// TwinCAT 3 PLC project PLC
// ProgramVersion: 3.1.4023.0
// libraries:
//   Tc2_Standard, * (Beckhoff Automation GmbH)
//   Tc2_System, * (Beckhoff Automation GmbH)
//   Tc3_Module, * (Beckhoff Automation GmbH)
// project tree:
//   / PlcTask.TcTTO
//   POUs/ MAIN.TcPOU
// real-time tasks:
//   TASK PlcTask: cycle T#4ms, priority 20, ADS port 350
// I/O:
//   DEVICE Device 1 (Profinet Controller), AmsNetId 5.24.131.22.2.1
//     tcpniodevice [Beckhoff Automation TwinCAT PLC PROFINET I/O Device with I/Os, V2.32, 1 port diagnostic supported TwinCAT PN Device]
//       modules: Term 1 (DAP Module), Term 2 (32 Byte In- and Output)
//   DEVICE Device 2 (TC3 EIP Scanner), AmsNetId 5.24.131.22.3.1
//     Box 2 (TC EtherNet/IP Slave) // <INFO> 172.16.17.2, Box 2 (TC EtherNet/IP Slave) (ProdCode: 6280, Rev: 3.01, Mac: 02:00:02:22:78:9c) </INFO> <EDS> C:\TwinCAT\3.1\Config\Io\EtherNetIP\TF6280.eds </EDS>
// variable links:
//   PLC Instance <-> Device 1 (Profinet Controller)/tcpniodevice
//     PlcTask Inputs/MAIN.arPNIn[{0..31}] <-> API/Term 2 (32 Byte In- and Output)/Subterm 4 (32 Byte In- and Output)/Inputs/1 Byte Input[{0..31}]  (32 links)
//     PlcTask Outputs/MAIN.arPNOut[{0..31}] <-> API/Term 2 (32 Byte In- and Output)/Subterm 4 (32 Byte In- and Output)/Outputs/1 Byte Output[{0..31}]  (32 links)
//   PLC Instance <-> Device 2 (TC3 EIP Scanner)/Box 2 (TC EtherNet/IP Slave)
//     PlcTask Inputs/MAIN.arEIPIn[{0..31}] <-> Connection 1 (Input/Output)/Inputs/data[{0..31}]  (32 links)
//     PlcTask Outputs/MAIN.arEIPOut[{0..31}] <-> Connection 1 (Input/Output)/Outputs/Var 239[{0..31}]  (32 links)

CONFIGURATION PLC
    RESOURCE PLC ON TwinCAT3
        TASK PlcTask(INTERVAL := T#4ms, PRIORITY := 20);
        PROGRAM MAIN WITH PlcTask : MAIN;
    END_RESOURCE
END_CONFIGURATION

// ---- POUs/MAIN.TcPOU
PROGRAM MAIN
VAR

	arGatewayIn					:ARRAY[0..31] OF BYTE;
    arGatewayOut				:ARRAY[0..31] OF BYTE;

	arPNIn				AT%I*	:ARRAY[0..31] OF BYTE;
	arPNOut				AT%Q*	:ARRAY[0..31] OF BYTE;	

	arEIPIn				AT%I*	:ARRAY[0..31] OF BYTE;
	arEIPOut			AT%Q*	:ARRAY[0..31] OF BYTE;
	
    {IF defined (PN)}
        sVariantUsed             :STRING := 'PN';	
    {ELSIF defined (EIP)}        
        sVariantUsed             :STRING := 'EIP';
    {END_IF}	

END_VAR



{IF defined (PN)}
  	arGatewayIn :=arPNIn;
{ELSIF defined (EIP)}
    arGatewayIn := arEIPIn;
{END_IF}

	arGatewayOut:=arGatewayIn;
	arEIPOut	:=arGatewayOut;
	arPNOut		:=arGatewayOut;

END_PROGRAM
